RoboDK station: Tarea3Definitiva_IsabellaCeballos.rdk

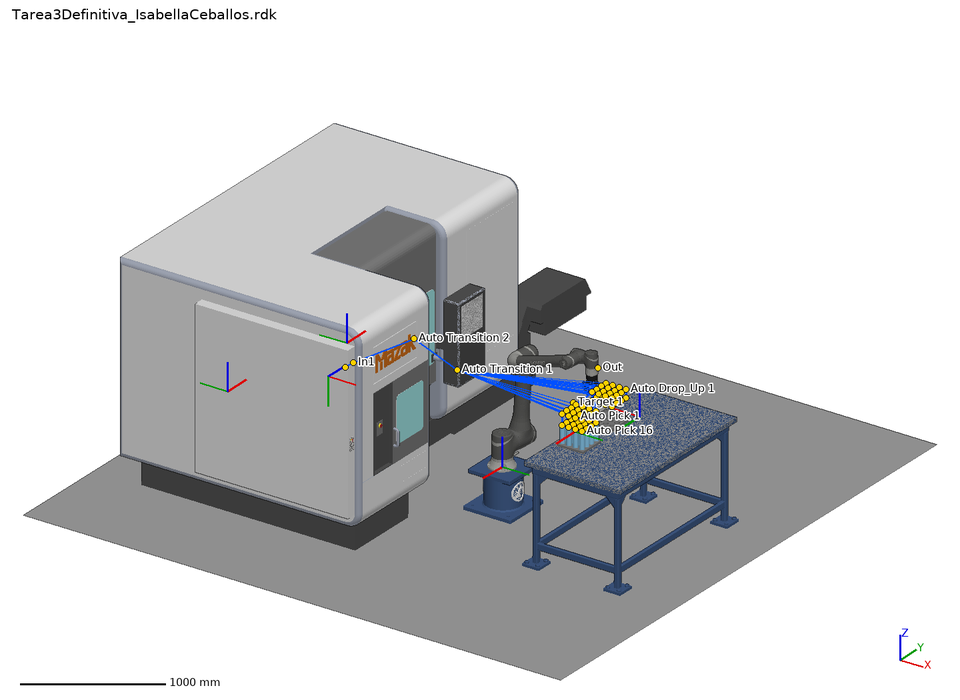
[picture v0: the station drawn from its stored meshes, robots at their saved joint values, targets as dots, program paths as lines]
Station Tarea3Definitiva_IsabellaCeballos (saved by RoboDK 5.5.1). Poses are relative to the parent item; angles as X-Y-Z fixed-axis rotations.
Station parameters (name, value as stored): TAGS, ['Machine Tending', 'CNC']
  - frame Omron TM12X Base at (300, 0, 70) mm, rotated rx 0 ry 0 rz -90 deg
    - robot Omron TM12X: 6 axes, payload 12 kg, reach 1300 mm, repeatability 0.1 mm, weight 33.3 kg
        modified DH rows (alpha deg, a mm, theta deg, d mm): 0, 0, 0, 165.2; 90, 0, 90, 0; 0, 636.1, 0, 0; 0, 557.9, -90, 156.3; -90, 0, 0, 106; 90, 0, 180, 113.15
        joint limits [-360, -360, -163, -360, -360, -360] to [360, 360, 163, 360, 360, 360]; home [0, 0, 90, -90, 90, 0]; saved at [263.092, -4.372, -66.936, -16.053, -91.349, 242.565]
      - tool g1, TCP at (0, 0, 130) mm, size 134.4 x 157.6 x 75 mm
      - tool RobotiQ 2F-85 Gripper (Open), TCP at (0, 0, 130) mm, size 147.4 x 146.8 x 75 mm
    - object Pedestal H12in (Type 1) at (0, 10, -300) mm, size 400 x 400 x 304.8 mm, geometry from Pedestal-H12in-Type-1.sld
  - frame Mazak Lathe Base at (-1000, 0, 650) mm, rotated rx 0 ry 0 rz 90 deg
    - robot Mazak Lathe: 1 axes
        modified DH rows (alpha deg, a mm, theta deg, d mm): 0, 0, 0, 0 linear
        base shift (0, 0, 0) mm, rotated rx 0 ry 90 rz 0 deg
        joint limits [0] to [700]; home [0]; saved at [0]
    - frame Lathe at (-368.68, -104.77, -79.13) mm, rotated rx -90 ry 0 rz -90 deg
  - frame Input at (1010, -140, 590) mm, rotated rx 0 ry 0 rz -90 deg
    - object Part Matrix at (0, 0, 0) mm, size 220 x 220 x 25 mm, geometry from Part Matrix.step
    - target Target 1 (Cartesian target) at (-26.53, -36.52, 202.61) mm, rotated rx -177.37 ry 1.91 rz -69.45 deg; joints [247.43, -1, -72.52, -13.29, -90.61, 226.91] of Omron TM12X
    - target Home (Cartesian target) at (28, 28, 225) mm, rotated rx -177.37 ry 1.91 rz -69.45 deg; joints [245.421, -8.702, -61.622, -16.467, -90.498, 224.904] of Omron TM12X
    - target Out (Cartesian target) at (-404.5, -94.61, 298.15) mm, rotated rx 179.32 ry 1.81 rz -82.53 deg; joints [279.536, -58.254, 58.657, -88.574, -89.388, -87.935] of Omron TM12X
    - target Auto Transition 1 (Cartesian target) at (259.07, -803.97, 350.52) mm, rotated rx -177.59 ry 1.72 rz -69.47 deg; joints [142.43, 16.067, -68.876, -37.376, -87.042, 121.929] of Omron TM12X
    - target Auto Transition 2 (Cartesian target) at (28.12, -1329.27, 350.52) mm, rotated rx -177.59 ry 1.72 rz -69.47 deg; joints [90.435, -6.151, -48.82, -37.474, -88.325, 69.903] of Omron TM12X
    - target Auto Up_Pick 1 (Cartesian target) at (28, 28, 225) mm, rotated rx -177.59 ry 1.72 rz -69.47 deg; joints [89.633, 54.83, -20.514, -126.784, -88.359, 69.101] of Omron TM12X
    - target Auto Pick 1 (Cartesian target) at (28, 28, 135) mm, rotated rx -177.59 ry 1.72 rz -69.47 deg; joints [89.633, 68.297, -42.42, -118.345, -88.359, 69.101] of Omron TM12X
    - target Auto Drop_Up 1 (Cartesian target) at (-374.01, 165.11, 220.31) mm, rotated rx -177.59 ry 1.72 rz -69.47 deg; joints [275.549, -61.889, 39.003, -64.828, -91.887, 255.015] of Omron TM12X
    - target Auto Drop 1 (Cartesian target) at (-374.01, 165.11, 156.87) mm, rotated rx -177.59 ry 1.72 rz -69.47 deg; joints [275.549, -69.478, 50.406, -68.642, -91.887, 255.015] of Omron TM12X
    - target Auto Up_Pick 2 (Cartesian target) at (28, 84, 225) mm, rotated rx -177.59 ry 1.72 rz -69.47 deg; joints [247.124, -65.005, 54.457, -76.543, -90.571, 226.613] of Omron TM12X
    - target Auto Pick 2 (Cartesian target) at (28, 84, 135) mm, rotated rx -177.59 ry 1.72 rz -69.47 deg; joints [89.659, 63.935, -29.058, -127.345, -88.358, 69.127] of Omron TM12X
    - target Auto Drop_Up 2 (Cartesian target) at (-374.01, 109.11, 220.31) mm, rotated rx -177.59 ry 1.72 rz -69.47 deg; joints [275.923, -64.235, 48.589, -72.079, -91.902, 255.389] of Omron TM12X
    - target Auto Drop 2 (Cartesian target) at (-374.01, 109.11, 156.87) mm, rotated rx -177.59 ry 1.72 rz -69.47 deg; joints [275.923, -71.126, 58.555, -75.154, -91.902, 255.389] of Omron TM12X
    - target Auto Up_Pick 3 (Cartesian target) at (28, 140, 225) mm, rotated rx -177.59 ry 1.72 rz -69.47 deg; joints [248.612, -20.473, -46.151, -20.483, -90.647, 228.099] of Omron TM12X
    - target Auto Pick 3 (Cartesian target) at (28, 140, 135) mm, rotated rx -177.59 ry 1.72 rz -69.47 deg; joints [248.612, -17.359, -60.205, -9.544, -90.647, 228.099] of Omron TM12X
    - target Auto Drop_Up 3 (Cartesian target) at (-374.01, 53.11, 220.31) mm, rotated rx -177.59 ry 1.72 rz -69.47 deg; joints [276.351, -13.266, -56.317, -18.157, -91.918, 255.817] of Omron TM12X
    - target Auto Drop 3 (Cartesian target) at (-374.01, 53.11, 156.87) mm, rotated rx -177.59 ry 1.72 rz -69.47 deg; joints [276.351, -11.379, -65.492, -10.869, -91.918, 255.817] of Omron TM12X
    - target Auto Up_Pick 4 (Cartesian target) at (28, 196, 225) mm, rotated rx -177.59 ry 1.72 rz -69.47 deg; joints [249.92, -27.448, -35.607, -24.068, -90.713, 229.405] of Omron TM12X
    - target Auto Pick 4 (Cartesian target) at (28, 196, 135) mm, rotated rx -177.59 ry 1.72 rz -69.47 deg; joints [249.92, -23.266, -51.89, -11.967, -90.713, 229.405] of Omron TM12X
    - target Auto Drop_Up 4 (Cartesian target) at (-374.01, -2.89, 220.31) mm, rotated rx -177.59 ry 1.72 rz -69.47 deg; joints [276.844, -7.931, -62.838, -16.988, -91.938, 256.31] of Omron TM12X
    - target Auto Drop 4 (Cartesian target) at (-374.01, -2.89, 156.87) mm, rotated rx -177.59 ry 1.72 rz -69.47 deg; joints [276.844, -6.251, -71.535, -9.971, -91.938, 256.31] of Omron TM12X
    - target Auto Up_Pick 5 (Cartesian target) at (84, 28, 225) mm, rotated rx -177.59 ry 1.72 rz -69.47 deg; joints [241.515, -10.232, -59.727, -17.09, -90.285, 221.011] of Omron TM12X
    - target Auto Pick 5 (Cartesian target) at (84, 28, 135) mm, rotated rx -177.59 ry 1.72 rz -69.47 deg; joints [241.515, -7.928, -72.043, -7.078, -90.285, 221.011] of Omron TM12X
    - target Auto Drop_Up 5 (Cartesian target) at (-318.01, 165.11, 220.31) mm, rotated rx -177.59 ry 1.72 rz -69.47 deg; joints [271.898, -23.816, -41.661, -22.121, -91.737, 251.365] of Omron TM12X
    - target Auto Drop 5 (Cartesian target) at (-318.01, 165.11, 156.87) mm, rotated rx -177.59 ry 1.72 rz -69.47 deg; joints [271.898, -21.097, -52.602, -13.899, -91.737, 251.365] of Omron TM12X
    - target Auto Up_Pick 6 (Cartesian target) at (84, 84, 225) mm, rotated rx -177.59 ry 1.72 rz -69.47 deg; joints [243.439, -15.802, -52.626, -18.633, -90.383, 222.933] of Omron TM12X
    - target Auto Pick 6 (Cartesian target) at (84, 84, 135) mm, rotated rx -177.59 ry 1.72 rz -69.47 deg; joints [243.439, -13.143, -65.721, -8.197, -90.383, 222.933] of Omron TM12X
    - target Auto Drop_Up 6 (Cartesian target) at (-318.01, 109.11, 220.31) mm, rotated rx -177.59 ry 1.72 rz -69.47 deg; joints [272.028, -17.436, -50.827, -19.34, -91.743, 251.496] of Omron TM12X
    - target Auto Drop 6 (Cartesian target) at (-318.01, 109.11, 156.87) mm, rotated rx -177.59 ry 1.72 rz -69.47 deg; joints [272.028, -15.303, -60.532, -11.766, -91.743, 251.496] of Omron TM12X
    - target Auto Up_Pick 7 (Cartesian target) at (84, 140, 225) mm, rotated rx -177.59 ry 1.72 rz -69.47 deg; joints [245.126, -21.925, -44.052, -21.096, -90.47, 224.618] of Omron TM12X
    - target Auto Pick 7 (Cartesian target) at (84, 140, 135) mm, rotated rx -177.59 ry 1.72 rz -69.47 deg; joints [245.126, -18.635, -58.475, -9.964, -90.47, 224.618] of Omron TM12X
    - target Auto Drop_Up 7 (Cartesian target) at (-318.01, 53.11, 220.31) mm, rotated rx -177.59 ry 1.72 rz -69.47 deg; joints [272.178, -11.695, -58.327, -17.585, -91.749, 251.645] of Omron TM12X
    - target Auto Drop 7 (Cartesian target) at (-318.01, 53.11, 156.87) mm, rotated rx -177.59 ry 1.72 rz -69.47 deg; joints [272.178, -9.884, -67.335, -10.387, -91.749, 251.645] of Omron TM12X
    - target Auto Up_Pick 8 (Cartesian target) at (84, 196, 225) mm, rotated rx -177.59 ry 1.72 rz -69.47 deg; joints [246.616, -29.108, -32.944, -25.035, -90.546, 226.106] of Omron TM12X
    - target Auto Pick 8 (Cartesian target) at (84, 196, 135) mm, rotated rx -177.59 ry 1.72 rz -69.47 deg; joints [246.616, -24.578, -49.957, -12.552, -90.546, 226.106] of Omron TM12X
    - target Auto Drop_Up 8 (Cartesian target) at (-318.01, -2.89, 220.31) mm, rotated rx -177.59 ry 1.72 rz -69.47 deg; joints [272.351, -6.333, -64.704, -16.575, -91.756, 251.819] of Omron TM12X
    - target Auto Drop 8 (Cartesian target) at (-318.01, -2.89, 156.87) mm, rotated rx -177.59 ry 1.72 rz -69.47 deg; joints [272.351, -4.699, -73.288, -9.625, -91.756, 251.819] of Omron TM12X
    - target Auto Up_Pick 9 (Cartesian target) at (140, 28, 225) mm, rotated rx -177.59 ry 1.72 rz -69.47 deg; joints [237.832, -12.037, -57.501, -17.499, -90.095, 217.333] of Omron TM12X
    - target Auto Pick 9 (Cartesian target) at (140, 28, 135) mm, rotated rx -177.59 ry 1.72 rz -69.47 deg; joints [237.832, -9.638, -70.034, -7.366, -90.095, 217.333] of Omron TM12X
    - target Auto Drop_Up 9 (Cartesian target) at (-262.01, 165.11, 220.31) mm, rotated rx -177.59 ry 1.72 rz -69.47 deg; joints [268.189, -22.573, -43.539, -21.379, -91.578, 247.658] of Omron TM12X
    - target Auto Drop 9 (Cartesian target) at (-262.01, 165.11, 156.87) mm, rotated rx -177.59 ry 1.72 rz -69.47 deg; joints [268.189, -19.996, -54.183, -13.312, -91.578, 247.658] of Omron TM12X
    - target Auto Up_Pick 10 (Cartesian target) at (140, 84, 225) mm, rotated rx -177.59 ry 1.72 rz -69.47 deg; joints [239.936, -17.62, -50.169, -19.254, -90.203, 219.434] of Omron TM12X
    - target Auto Pick 10 (Cartesian target) at (140, 84, 135) mm, rotated rx -177.59 ry 1.72 rz -69.47 deg; joints [239.936, -14.805, -63.596, -8.642, -90.203, 219.434] of Omron TM12X
    - target Auto Drop_Up 10 (Cartesian target) at (-262.01, 109.11, 220.31) mm, rotated rx -177.59 ry 1.72 rz -69.47 deg; joints [268.063, -16.266, -52.435, -18.786, -91.573, 247.532] of Omron TM12X
    - target Auto Drop 10 (Cartesian target) at (-262.01, 109.11, 156.87) mm, rotated rx -177.59 ry 1.72 rz -69.47 deg; joints [268.063, -14.216, -61.968, -11.304, -91.573, 247.532] of Omron TM12X
    - target Auto Up_Pick 11 (Cartesian target) at (140, 140, 225) mm, rotated rx -177.59 ry 1.72 rz -69.47 deg; joints [241.792, -23.852, -41.191, -22.008, -90.299, 221.288] of Omron TM12X
    - target Auto Pick 11 (Cartesian target) at (140, 140, 135) mm, rotated rx -177.59 ry 1.72 rz -69.47 deg; joints [241.792, -20.294, -56.173, -10.585, -90.299, 221.288] of Omron TM12X
    - target Auto Drop_Up 11 (Cartesian target) at (-262.01, 53.11, 220.31) mm, rotated rx -177.59 ry 1.72 rz -69.47 deg; joints [267.918, -10.535, -59.783, -17.165, -91.566, 247.387] of Omron TM12X
    - target Auto Drop 11 (Cartesian target) at (-262.01, 53.11, 156.87) mm, rotated rx -177.59 ry 1.72 rz -69.47 deg; joints [267.918, -8.774, -68.68, -10.029, -91.566, 247.387] of Omron TM12X
    - target Auto Up_Pick 12 (Cartesian target) at (140, 196, 225) mm, rotated rx -177.59 ry 1.72 rz -69.47 deg; joints [243.439, -31.4, -29.157, -26.504, -90.383, 222.933] of Omron TM12X
    - target Auto Pick 12 (Cartesian target) at (140, 196, 135) mm, rotated rx -177.59 ry 1.72 rz -69.47 deg; joints [243.439, -26.305, -47.355, -13.401, -90.383, 222.933] of Omron TM12X
    - target Auto Drop_Up 12 (Cartesian target) at (-262.01, -2.89, 220.31) mm, rotated rx -177.59 ry 1.72 rz -69.47 deg; joints [267.749, -5.144, -66.063, -16.272, -91.559, 247.219] of Omron TM12X
    - target Auto Drop 12 (Cartesian target) at (-262.01, -2.89, 156.87) mm, rotated rx -177.59 ry 1.72 rz -69.47 deg; joints [267.749, -3.538, -74.571, -9.369, -91.559, 247.219] of Omron TM12X
    - target Auto Up_Pick 13 (Cartesian target) at (196, 28, 225) mm, rotated rx -177.59 ry 1.72 rz -69.47 deg; joints [234.382, -14.253, -54.671, -18.113, -89.916, 213.888] of Omron TM12X
    - target Auto Pick 13 (Cartesian target) at (196, 28, 135) mm, rotated rx -177.59 ry 1.72 rz -69.47 deg; joints [234.382, -11.712, -67.515, -7.811, -89.916, 213.888] of Omron TM12X
    - target Auto Drop_Up 13 (Cartesian target) at (-206.01, 165.11, 220.31) mm, rotated rx -177.59 ry 1.72 rz -69.47 deg; joints [264.452, -21.782, -44.722, -20.889, -91.411, 243.923] of Omron TM12X
    - target Auto Drop 13 (Cartesian target) at (-206.01, 165.11, 156.87) mm, rotated rx -177.59 ry 1.72 rz -69.47 deg; joints [264.452, -19.29, -55.189, -12.914, -91.411, 243.923] of Omron TM12X
    - target Auto Up_Pick 14 (Cartesian target) at (196, 84, 225) mm, rotated rx -177.59 ry 1.72 rz -69.47 deg; joints [236.628, -19.883, -47.008, -20.145, -90.032, 216.131] of Omron TM12X
    - target Auto Pick 14 (Cartesian target) at (196, 84, 135) mm, rotated rx -177.59 ry 1.72 rz -69.47 deg; joints [236.628, -16.839, -60.917, -9.28, -90.032, 216.131] of Omron TM12X
    - target Auto Drop_Up 14 (Cartesian target) at (-206.01, 109.11, 220.31) mm, rotated rx -177.59 ry 1.72 rz -69.47 deg; joints [264.063, -15.515, -53.458, -18.41, -91.394, 243.534] of Omron TM12X
    - target Auto Drop 14 (Cartesian target) at (-206.01, 109.11, 156.87) mm, rotated rx -177.59 ry 1.72 rz -69.47 deg; joints [264.063, -13.514, -62.887, -10.982, -91.394, 243.534] of Omron TM12X
    - target Auto Up_Pick 15 (Cartesian target) at (196, 140, 225) mm, rotated rx -177.59 ry 1.72 rz -69.47 deg; joints [238.622, -26.311, -37.416, -23.312, -90.135, 218.122] of Omron TM12X
    - target Auto Pick 15 (Cartesian target) at (196, 140, 135) mm, rotated rx -177.59 ry 1.72 rz -69.47 deg; joints [238.622, -22.348, -53.243, -11.448, -90.135, 218.122] of Omron TM12X
    - target Auto Drop_Up 15 (Cartesian target) at (-206.01, 53.11, 220.31) mm, rotated rx -177.59 ry 1.72 rz -69.47 deg; joints [263.614, -9.785, -60.715, -16.873, -91.373, 243.087] of Omron TM12X
    - target Auto Drop 15 (Cartesian target) at (-206.01, 53.11, 156.87) mm, rotated rx -177.59 ry 1.72 rz -69.47 deg; joints [263.614, -8.054, -69.544, -9.775, -91.373, 243.087] of Omron TM12X
    - target Auto Up_Pick 16 (Cartesian target) at (196, 196, 225) mm, rotated rx -177.59 ry 1.72 rz -69.47 deg; joints [240.402, -34.545, -23.748, -28.751, -90.227, 219.899] of Omron TM12X
    - target Auto Pick 16 (Cartesian target) at (196, 196, 135) mm, rotated rx -177.59 ry 1.72 rz -69.47 deg; joints [240.402, -28.482, -43.987, -14.576, -90.227, 219.899] of Omron TM12X
    - target Auto Drop_Up 16 (Cartesian target) at (-206.01, -2.89, 220.31) mm, rotated rx -177.59 ry 1.72 rz -69.47 deg; joints [263.092, -4.372, -66.936, -16.053, -91.349, 242.565] of Omron TM12X
    - target Auto Drop 16 (Cartesian target) at (-206.01, -2.89, 156.87) mm, rotated rx -177.59 ry 1.72 rz -69.47 deg; joints [263.092, -2.783, -75.398, -9.18, -91.349, 242.565] of Omron TM12X
    - object Part 14 at (27.5, 137.5, -20) mm, size 40 x 40 x 150 mm, geometry from Part.step
    - object Part 13 at (27.5, 192.5, -20) mm, size 40 x 40 x 150 mm, geometry from Part.step
    - object Part 11 at (82.5, 82.5, -20) mm, size 40 x 40 x 150 mm, geometry from Part.step
    - object Part 10 at (82.5, 137.5, -20) mm, size 40 x 40 x 150 mm, geometry from Part.step
    - object Part 9 at (82.5, 192.5, -20) mm, size 40 x 40 x 150 mm, geometry from Part.step
    - object Part 8 at (137.5, 27.5, -20) mm, size 40 x 40 x 150 mm, geometry from Part.step
    - object Part 6 at (137.5, 137.5, -20) mm, size 40 x 40 x 150 mm, geometry from Part.step
    - object Part 1 at (192.5, 192.5, -20) mm, size 40 x 40 x 150 mm, geometry from Part.step
    - object Part 16 at (27.5, 27.5, -20) mm, size 40 x 40 x 150 mm, geometry from Part.step
    - object Part 12 at (82.5, 27.5, -20) mm, size 40 x 40 x 150 mm, geometry from Part.step
    - object Part 5 at (137.5, 192.5, -20) mm, size 40 x 40 x 150 mm, geometry from Part.step
    - object Part 7 at (137.5, 82.5, -20) mm, size 40 x 40 x 150 mm, geometry from Part.step
    - object Part 4 at (192.5, 27.5, -20) mm, rotated rx 0 ry 0 rz -180 deg, size 40 x 40 x 150 mm, geometry from Part.step
    - object Part 3 at (192.5, 82.5, -20) mm, rotated rx 0 ry 0 rz -180 deg, size 40 x 40 x 150 mm, geometry from Part.step
    - object Part 2 at (192.5, 137.5, -20) mm, rotated rx 0 ry 0 rz -180 deg, size 40 x 40 x 150 mm, geometry from Part.step
    - object Part 15 at (27.5, 82.5, -20) mm, size 40 x 40 x 150 mm, geometry from Part.step
  - frame Output at (1250, 290, 600) mm, rotated rx 0 ry 0 rz -180 deg
    - object Part Matrix at (47.8, 28.1, 0) mm, size 220 x 220 x 25 mm, geometry from Part Matrix.step
  - frame World at (-2000, 0, 0) mm, rotated rx 0 ry 0 rz 90 deg
    - object Floor at (250, -1940, -230) mm, size 4500 x 4500 x 0 mm, geometry from Floor (2).sld
    - object Table 1400x800x800mm at (-340, -3360, 570) mm, size 1420 x 820 x 800 mm, geometry from Table-1400x800x800mm.sld
    - target OpenDoor (Cartesian target) at (700, -1000, 650) mm; joints [700] of Mazak Lathe
    - target CloseDoor (Cartesian target) at (0, -1000, 650) mm; joints [0] of Mazak Lathe
    - target In1 (Cartesian target) at (-137.95, -1150.25, 595.88) mm, rotated rx -86.34 ry 2.11 rz 94.34 deg; joints [77.244, -89.992, 25.646, 51.981, -342.661, 170.292] of Omron TM12X
    - target In2 (Cartesian target) at (-206.56, -1130.76, 584.67) mm, rotated rx -87.8 ry 7.87 rz 92.76 deg; joints [-84.147, 66.082, 6.025, 75.079, -175.968, 40.623] of Omron TM12X
  - Python program Main_Program_Python (listed below)
  - program atach (1 instructions, listed below)
  - program detach (1 instructions, listed below)
  - program init (1 instructions, listed below)
  - program OpenDoor (2 instructions, listed below)
  - program CloseDoor (2 instructions, listed below)
  - program GoHome (3 instructions, listed below)
  - program Go_Out (3 instructions, listed below)
  - program Main_Program (496 instructions, listed below)
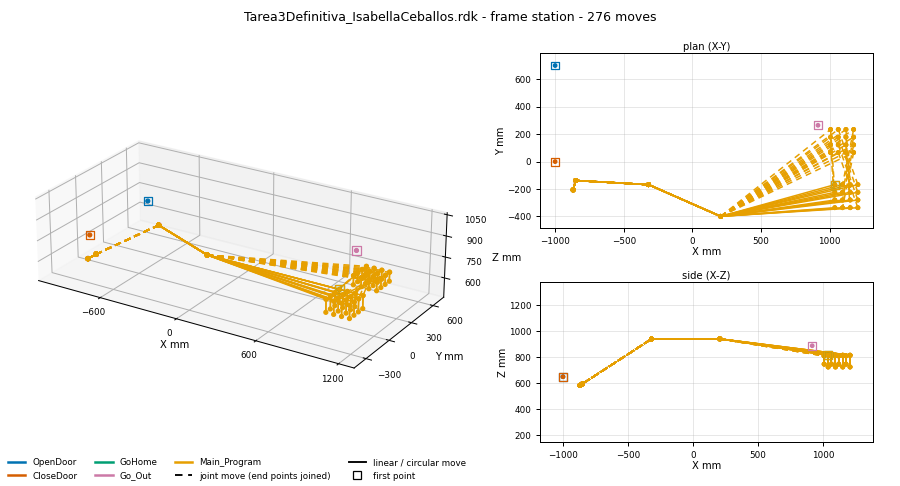
[picture p0: tool path of Tarea3Definitiva_IsabellaCeballos.rdk in frame station, 276 of 276 moves have a stored position in this frame; points joined in program order, loops and branches not executed]

--- Python program Main_Program_Python ---
from robolink import *    # Robot toolbox
import time as t

# Link to RoboDK
RDK = Robolink() # Interactuar con la interfaz del robot

# Mecanismos
robot = RDK.Item("Omron TM12X", ITEM_TYPE_ROBOT) #Robot
MAZAK = RDK.Item("Mazak Lathe") # Mazak
Tool_gripper = RDK.Item('g1',ITEM_TYPE_TOOL ) #Gripper

#Esto es para que no se repitan cosas en el código
list_names = RDK.ItemList(None, True)
for item_name in list_names:
    if item_name.startswith('Auto'):
        RDK.Item(item_name).Delete()
    if item_name.startswith('Main_'):
        RDK.Item(item_name).Delete()

#Código para generar puntos de botellas
def gridXY (m,n,d, e):

    """
     m= número de puntos en x
     n= número de puntos en y
     d= distancia entre cada punto en m

     En este ejercicio m = n, es cuadrado el soporte. 4x4
    """

    lista_puntos = []
    coeficientes = [1, 3, 5, 7 ]
    for i in range(m):
        for j in range(n):
            punto = [coeficientes[i]*d, coeficientes[j]*e, 225.000]
            lista_puntos.append(punto)


    return lista_puntos

m = 4
n = 4
d = 28
e = 28


puntos = gridXY(m,n,d,e)


# Código Principal

# Marcos de referencias
Input = RDK.Item("Input",ITEM_TYPE_FRAME) #frame
Output = RDK.Item("Output",ITEM_TYPE_FRAME)#frame2
Lathe = RDK.Item("Lathe",ITEM_TYPE_FRAME) #frame3
World = RDK.Item("World",ITEM_TYPE_FRAME) #frame4



robot.setPoseFrame(Input) #asociamos el robot a Input
pose_ref = robot.Pose()

Program = RDK.AddProgram('Main_Program')# Se genera programa


j = 0

#TARGETS DEL PROGRAMA

In1 = RDK.Item('In1',ITEM_TYPE_TARGET)
In2 = RDK.Item('In2',ITEM_TYPE_TARGET)
In3 = RDK.Item('In3',ITEM_TYPE_TARGET)


robot.setPoseFrame(Input)

    #TRANSITION 1
Trans1 = RDK.AddTarget('Auto Transition 1')#ti7
pose_t = pose_ref
pose_t.setPos([259.072, -803.965, 350.521] )
Trans1.setPose(pose_t)
Trans1.setAsCartesianTarget()
Trans1.setVisible(0)

    #TRANSITION 2
Trans2 = RDK.AddTarget('Auto Transition 2') #ti9
pose_t.setPos([28.119, -1329.271, 350.521] )
Trans2.setPose(pose_t)
Trans2.setAsCartesianTarget()
Trans2.setVisible(0)

# Funciones del programa

def Pick_up(P,Pick_Up,Pick):
    P.MoveJ(Pick_Up)
    t.sleep(0.5)
    P.MoveL(Pick)
    t.sleep(0.5)
    P.RunInstruction('atach',0)
    t.sleep(0.5)
    P.MoveL(Pick_Up)
    t.sleep(0.5)
    return

def Drop_out(P,Drop,Drop_Up):
    P.MoveJ(Drop_Up)
    t.sleep(0.5)
    P.MoveL(Drop)
    t.sleep(0.5)
    P.RunInstruction('detach',0)
    t.sleep(0.5)
    P.MoveL(Drop_Up)
    t.sleep(0.5)
    return

def Pick_Lathe_Transition(P,Trans1,Trans2):
    P.MoveL(Trans1)
    t.sleep(0.5)
    P.MoveJ(Trans2)
    t.sleep(0.5)
    return

def PickLathe(P,In1,In2,In3,Trans2):
    P.setFrame(World)
    P.MoveJ(In1)
    P.MoveL(In2)
    P.RunInstruction('detach',0)
    t.sleep(0.5)
    P.MoveL(In1)
    t.sleep(0.5)
    P.setFrame(Input)
    t.sleep(0.5)
    P.MoveJ(Trans2)
    t.sleep(5)
    return

def DropLathe(P,In1,In2,Trans2):
    P.setFrame(World)
    P.MoveJ(In1)
    P.MoveL(In2)
    P.RunInstruction('atach',0)
    t.sleep(0.5)
    P.MoveL(In1)
    t.sleep(0.5)
    P.setFrame(Input)
    t.sleep(0.5)
    P.MoveJ(Trans2)
    t.sleep(5)
    return


for i in puntos:

    #**GENARACIÓN DE TARGETS PICK BOTELLAS**
    #---------------------------------------
    robot.setPoseFrame(Input)
    Pick_Up = RDK.AddTarget('Auto Up_Pick %i' %(j+1))
    pose_i = pose_ref
    pose_i.setPos(i) #lista [x,y,z]
    Pick_Up.setPose(pose_i)
    Pick_Up.setAsCartesianTarget()
    Pick_Up.setVisible(0)
    #--------------------------------------
    Pick = RDK.AddTarget('Auto Pick %i' %(j+1))
    pose_j = pose_i
    pose_j.setPos([i[0],i[1], 135] )#[x,y,z]
    Pick.setPose(pose_j)
    Pick.setAsCartesianTarget()
    Pick.setVisible(0)



    #**GENERACIÓN DE TARGETS DROP BOTELLAS**
    #---------------------------------------
    Drop_Up = RDK.AddTarget('Auto Drop_Up %i' %(j+1))
    pose_p = pose_i
    pose_p.setPos([-402.010 + i[0], 193.114 - i[1], 220.306] )#[x,y,z]
    Drop_Up.setPose(pose_p)
    Drop_Up.setAsCartesianTarget()
    Drop_Up.setVisible(0)
   #---------------------------------------
    Drop = RDK.AddTarget('Auto Drop %i' %(j+1))
    pose_r = pose_i
    pose_r.setPos([-402.010 + i[0], 193.114 - i[1], 156.874] )#[x,y,z]
    Drop.setPose(pose_r)
    Drop.setAsCartesianTarget()
    Drop.setVisible(0)



    # SECUENCIA
    Program.setFrame(Input)
    Pick_up(Program,Pick_Up,Pick)
    Pick_Lathe_Transition(Program,Trans1,Trans2)
    Program.RunInstruction('OpenDoor',0)
    PickLathe(Program,In1,In2,In3,Trans2)
    Program.RunInstruction('CloseDoor',0)
    Program.RunInstruction('OpenDoor',0)
    DropLathe(Program,In1,In2,Trans2)
    Program.RunInstruction('CloseDoor',0)
    Program.MoveL(Trans1)
    Program.RunInstruction('Go_Out',0)
    Drop_out(Program,Drop,Drop_Up)


    j+=1

--- program atach (robot Omron TM12X) ---
  Adjuntar a g1

--- program detach (robot Omron TM12X) ---
  Separar de g1

--- program init (robot Omron TM12X) ---
  Reemplazar objetos

--- program OpenDoor (robot Mazak Lathe) ---
  Est. Ref.: World
  MoveJ (OpenDoor)

--- program CloseDoor (robot Mazak Lathe) ---
  Est. Ref.: World
  MoveJ (CloseDoor)

--- program GoHome (robot Omron TM12X) ---
  Est. Ref.: Input
  Est. herr: g1
  MoveJ (Home)

--- program Go_Out (robot Omron TM12X) ---
  Est. Ref.: Input
  Est. herr: g1
  MoveJ (Out)

--- program Main_Program (robot Omron TM12X) ---
  Est. Ref.: Input
  MoveJ (Auto Up_Pick 1)
  MoveL (Auto Pick 1)
  Llamar atach
  MoveL (Auto Up_Pick 1)
  MoveL (Auto Transition 1)
  MoveJ (Auto Transition 2)
  Llamar OpenDoor
  Est. Ref.: World
  MoveJ (In1)
  MoveL (In2)
  Llamar detach
  MoveL (In1)
  Est. Ref.: Input
  MoveJ (Auto Transition 2)
  Llamar CloseDoor
  Llamar OpenDoor
  Est. Ref.: World
  MoveJ (In1)
  MoveL (In2)
  Llamar atach
  MoveL (In1)
  Est. Ref.: Input
  MoveJ (Auto Transition 2)
  Llamar CloseDoor
  MoveL (Auto Transition 1)
  Llamar Go_Out
  MoveJ (Auto Drop_Up 1)
  MoveL (Auto Drop 1)
  Llamar detach
  MoveL (Auto Drop_Up 1)
  Est. Ref.: Input
  MoveJ (Auto Up_Pick 2)
  MoveL (Auto Pick 2)
  Llamar atach
  MoveL (Auto Up_Pick 2)
  MoveL (Auto Transition 1)
  MoveJ (Auto Transition 2)
  Llamar OpenDoor
  Est. Ref.: World
  MoveJ (In1)
  MoveL (In2)
  Llamar detach
  MoveL (In1)
  Est. Ref.: Input
  MoveJ (Auto Transition 2)
  Llamar CloseDoor
  Llamar OpenDoor
  Est. Ref.: World
  MoveJ (In1)
  MoveL (In2)
  Llamar atach
  MoveL (In1)
  Est. Ref.: Input
  MoveJ (Auto Transition 2)
  Llamar CloseDoor
  MoveL (Auto Transition 1)
  Llamar Go_Out
  MoveJ (Auto Drop_Up 2)
  MoveL (Auto Drop 2)
  Llamar detach
  MoveL (Auto Drop_Up 2)
  Est. Ref.: Input
  MoveJ (Auto Up_Pick 3)
  MoveL (Auto Pick 3)
  Llamar atach
  MoveL (Auto Up_Pick 3)
  MoveL (Auto Transition 1)
  MoveJ (Auto Transition 2)
  Llamar OpenDoor
  Est. Ref.: World
  MoveJ (In1)
  MoveL (In2)
  Llamar detach
  MoveL (In1)
  Est. Ref.: Input
  MoveJ (Auto Transition 2)
  Llamar CloseDoor
  Llamar OpenDoor
  Est. Ref.: World
  MoveJ (In1)
  MoveL (In2)
  Llamar atach
  MoveL (In1)
  Est. Ref.: Input
  MoveJ (Auto Transition 2)
  Llamar CloseDoor
  MoveL (Auto Transition 1)
  Llamar Go_Out
  MoveJ (Auto Drop_Up 3)
  MoveL (Auto Drop 3)
  Llamar detach
  MoveL (Auto Drop_Up 3)
  Est. Ref.: Input
  MoveJ (Auto Up_Pick 4)
  MoveL (Auto Pick 4)
  Llamar atach
  MoveL (Auto Up_Pick 4)
  MoveL (Auto Transition 1)
  MoveJ (Auto Transition 2)
  Llamar OpenDoor
  Est. Ref.: World
  MoveJ (In1)
  MoveL (In2)
  Llamar detach
  MoveL (In1)
  Est. Ref.: Input
  MoveJ (Auto Transition 2)
  Llamar CloseDoor
  Llamar OpenDoor
  Est. Ref.: World
  MoveJ (In1)
  MoveL (In2)
  Llamar atach
  MoveL (In1)
  Est. Ref.: Input
  MoveJ (Auto Transition 2)
  Llamar CloseDoor
  MoveL (Auto Transition 1)
  Llamar Go_Out
  MoveJ (Auto Drop_Up 4)
  MoveL (Auto Drop 4)
  Llamar detach
  MoveL (Auto Drop_Up 4)
  Est. Ref.: Input
  MoveJ (Auto Up_Pick 5)
  MoveL (Auto Pick 5)
  Llamar atach
  MoveL (Auto Up_Pick 5)
  MoveL (Auto Transition 1)
  MoveJ (Auto Transition 2)
  Llamar OpenDoor
  Est. Ref.: World
  MoveJ (In1)
  MoveL (In2)
  Llamar detach
  MoveL (In1)
  Est. Ref.: Input
  MoveJ (Auto Transition 2)
  Llamar CloseDoor
  Llamar OpenDoor
  Est. Ref.: World
  MoveJ (In1)
  MoveL (In2)
  Llamar atach
  MoveL (In1)
  Est. Ref.: Input
  MoveJ (Auto Transition 2)
  Llamar CloseDoor
  MoveL (Auto Transition 1)
  Llamar Go_Out
  MoveJ (Auto Drop_Up 5)
  MoveL (Auto Drop 5)
  Llamar detach
  MoveL (Auto Drop_Up 5)
  Est. Ref.: Input
  MoveJ (Auto Up_Pick 6)
  MoveL (Auto Pick 6)
  Llamar atach
  MoveL (Auto Up_Pick 6)
  MoveL (Auto Transition 1)
  MoveJ (Auto Transition 2)
  Llamar OpenDoor
  Est. Ref.: World
  MoveJ (In1)
  MoveL (In2)
  Llamar detach
  MoveL (In1)
  Est. Ref.: Input
  MoveJ (Auto Transition 2)
  Llamar CloseDoor
  Llamar OpenDoor
  Est. Ref.: World
  MoveJ (In1)
  MoveL (In2)
  Llamar atach
  MoveL (In1)
  Est. Ref.: Input
  MoveJ (Auto Transition 2)
  Llamar CloseDoor
  MoveL (Auto Transition 1)
  Llamar Go_Out
  MoveJ (Auto Drop_Up 6)
  MoveL (Auto Drop 6)
  Llamar detach
  MoveL (Auto Drop_Up 6)
  Est. Ref.: Input
  MoveJ (Auto Up_Pick 7)
  MoveL (Auto Pick 7)
  Llamar atach
  MoveL (Auto Up_Pick 7)
  MoveL (Auto Transition 1)
  MoveJ (Auto Transition 2)
  Llamar OpenDoor
  Est. Ref.: World
  MoveJ (In1)
  MoveL (In2)
  Llamar detach
  MoveL (In1)
  Est. Ref.: Input
  MoveJ (Auto Transition 2)
  Llamar CloseDoor
  Llamar OpenDoor
  Est. Ref.: World
  MoveJ (In1)
  MoveL (In2)
  Llamar atach
  MoveL (In1)
  Est. Ref.: Input
  MoveJ (Auto Transition 2)
  Llamar CloseDoor
  MoveL (Auto Transition 1)
  Llamar Go_Out
  MoveJ (Auto Drop_Up 7)
  MoveL (Auto Drop 7)
  Llamar detach
  MoveL (Auto Drop_Up 7)
  Est. Ref.: Input
  MoveJ (Auto Up_Pick 8)
  MoveL (Auto Pick 8)
  Llamar atach
  MoveL (Auto Up_Pick 8)
  MoveL (Auto Transition 1)
  MoveJ (Auto Transition 2)
  Llamar OpenDoor
  Est. Ref.: World
  MoveJ (In1)
  MoveL (In2)
  Llamar detach
  MoveL (In1)
  Est. Ref.: Input
  MoveJ (Auto Transition 2)
  Llamar CloseDoor
  Llamar OpenDoor
  Est. Ref.: World
  MoveJ (In1)
  MoveL (In2)
  Llamar atach
  MoveL (In1)
  Est. Ref.: Input
  MoveJ (Auto Transition 2)
  Llamar CloseDoor
  MoveL (Auto Transition 1)
  Llamar Go_Out
  MoveJ (Auto Drop_Up 8)
  MoveL (Auto Drop 8)
  Llamar detach
  MoveL (Auto Drop_Up 8)
  Est. Ref.: Input
  MoveJ (Auto Up_Pick 9)
  MoveL (Auto Pick 9)
  Llamar atach
  MoveL (Auto Up_Pick 9)
  MoveL (Auto Transition 1)
  MoveJ (Auto Transition 2)
  Llamar OpenDoor
  Est. Ref.: World
  MoveJ (In1)
  MoveL (In2)
  Llamar detach
  MoveL (In1)
  Est. Ref.: Input
  MoveJ (Auto Transition 2)
  Llamar CloseDoor
  Llamar OpenDoor
  Est. Ref.: World
  MoveJ (In1)
  MoveL (In2)
  Llamar atach
  MoveL (In1)
  Est. Ref.: Input
  MoveJ (Auto Transition 2)
  Llamar CloseDoor
  MoveL (Auto Transition 1)
  Llamar Go_Out
  MoveJ (Auto Drop_Up 9)
  MoveL (Auto Drop 9)
  Llamar detach
  MoveL (Auto Drop_Up 9)
  Est. Ref.: Input
  MoveJ (Auto Up_Pick 10)
  MoveL (Auto Pick 10)
  Llamar atach
  MoveL (Auto Up_Pick 10)
  MoveL (Auto Transition 1)
  MoveJ (Auto Transition 2)
  Llamar OpenDoor
  Est. Ref.: World
  MoveJ (In1)
  MoveL (In2)
  Llamar detach
  MoveL (In1)
  Est. Ref.: Input
  MoveJ (Auto Transition 2)
  Llamar CloseDoor
  Llamar OpenDoor
  Est. Ref.: World
  MoveJ (In1)
  MoveL (In2)
  Llamar atach
  MoveL (In1)
  Est. Ref.: Input
  MoveJ (Auto Transition 2)
  Llamar CloseDoor
  MoveL (Auto Transition 1)
  Llamar Go_Out
  MoveJ (Auto Drop_Up 10)
  MoveL (Auto Drop 10)
  Llamar detach
  MoveL (Auto Drop_Up 10)
  Est. Ref.: Input
  MoveJ (Auto Up_Pick 11)
  MoveL (Auto Pick 11)
  Llamar atach
  MoveL (Auto Up_Pick 11)
  MoveL (Auto Transition 1)
  MoveJ (Auto Transition 2)
  Llamar OpenDoor
  Est. Ref.: World
  MoveJ (In1)
  MoveL (In2)
  Llamar detach
  MoveL (In1)
  Est. Ref.: Input
  MoveJ (Auto Transition 2)
  Llamar CloseDoor
  Llamar OpenDoor
  Est. Ref.: World
  MoveJ (In1)
  MoveL (In2)
  Llamar atach
  MoveL (In1)
  Est. Ref.: Input
  MoveJ (Auto Transition 2)
  Llamar CloseDoor
  MoveL (Auto Transition 1)
  Llamar Go_Out
  MoveJ (Auto Drop_Up 11)
  MoveL (Auto Drop 11)
  Llamar detach
  MoveL (Auto Drop_Up 11)
  Est. Ref.: Input
  MoveJ (Auto Up_Pick 12)
  MoveL (Auto Pick 12)
  Llamar atach
  MoveL (Auto Up_Pick 12)
  MoveL (Auto Transition 1)
  MoveJ (Auto Transition 2)
  Llamar OpenDoor
  Est. Ref.: World
  MoveJ (In1)
  MoveL (In2)
  Llamar detach
  MoveL (In1)
  Est. Ref.: Input
  MoveJ (Auto Transition 2)
  Llamar CloseDoor
  Llamar OpenDoor
  Est. Ref.: World
  MoveJ (In1)
  MoveL (In2)
  Llamar atach
  MoveL (In1)
  Est. Ref.: Input
  MoveJ (Auto Transition 2)
  Llamar CloseDoor
  MoveL (Auto Transition 1)
  Llamar Go_Out
  MoveJ (Auto Drop_Up 12)
  MoveL (Auto Drop 12)
  Llamar detach
  MoveL (Auto Drop_Up 12)
  Est. Ref.: Input
  MoveJ (Auto Up_Pick 13)
  MoveL (Auto Pick 13)
  Llamar atach
  MoveL (Auto Up_Pick 13)
  MoveL (Auto Transition 1)
  MoveJ (Auto Transition 2)
  Llamar OpenDoor
  Est. Ref.: World
  MoveJ (In1)
  MoveL (In2)
  Llamar detach
  MoveL (In1)
  Est. Ref.: Input
  MoveJ (Auto Transition 2)
  Llamar CloseDoor
  Llamar OpenDoor
  Est. Ref.: World
  MoveJ (In1)
  MoveL (In2)
  Llamar atach
  MoveL (In1)
  Est. Ref.: Input
  MoveJ (Auto Transition 2)
  Llamar CloseDoor
  MoveL (Auto Transition 1)
  Llamar Go_Out
  MoveJ (Auto Drop_Up 13)
  MoveL (Auto Drop 13)
  Llamar detach
  MoveL (Auto Drop_Up 13)
  Est. Ref.: Input
  MoveJ (Auto Up_Pick 14)
  MoveL (Auto Pick 14)
  Llamar atach
  MoveL (Auto Up_Pick 14)
  MoveL (Auto Transition 1)
  MoveJ (Auto Transition 2)
  Llamar OpenDoor
  Est. Ref.: World
  MoveJ (In1)
  MoveL (In2)
  Llamar detach
  MoveL (In1)
  Est. Ref.: Input
  MoveJ (Auto Transition 2)
  Llamar CloseDoor
  Llamar OpenDoor
  Est. Ref.: World
  MoveJ (In1)
  MoveL (In2)
  Llamar atach
  MoveL (In1)
  Est. Ref.: Input
  MoveJ (Auto Transition 2)
  Llamar CloseDoor
  MoveL (Auto Transition 1)
  Llamar Go_Out
  MoveJ (Auto Drop_Up 14)
  MoveL (Auto Drop 14)
  Llamar detach
  MoveL (Auto Drop_Up 14)
  Est. Ref.: Input
  MoveJ (Auto Up_Pick 15)
  MoveL (Auto Pick 15)
  Llamar atach
  MoveL (Auto Up_Pick 15)
  MoveL (Auto Transition 1)
  MoveJ (Auto Transition 2)
  Llamar OpenDoor
  Est. Ref.: World
  MoveJ (In1)
  MoveL (In2)
  Llamar detach
  MoveL (In1)
  Est. Ref.: Input
  MoveJ (Auto Transition 2)
  Llamar CloseDoor
  Llamar OpenDoor
  Est. Ref.: World
  MoveJ (In1)
  MoveL (In2)
  Llamar atach
  MoveL (In1)
  Est. Ref.: Input
  MoveJ (Auto Transition 2)
  Llamar CloseDoor
  MoveL (Auto Transition 1)
  Llamar Go_Out
  MoveJ (Auto Drop_Up 15)
  MoveL (Auto Drop 15)
  Llamar detach
  MoveL (Auto Drop_Up 15)
  Est. Ref.: Input
  MoveJ (Auto Up_Pick 16)
  MoveL (Auto Pick 16)
  Llamar atach
  MoveL (Auto Up_Pick 16)
  MoveL (Auto Transition 1)
  MoveJ (Auto Transition 2)
  Llamar OpenDoor
  Est. Ref.: World
  MoveJ (In1)
  MoveL (In2)
  Llamar detach
  MoveL (In1)
  Est. Ref.: Input
  MoveJ (Auto Transition 2)
  Llamar CloseDoor
  Llamar OpenDoor
  Est. Ref.: World
  MoveJ (In1)
  MoveL (In2)
  Llamar atach
  MoveL (In1)
  Est. Ref.: Input
  MoveJ (Auto Transition 2)
  Llamar CloseDoor
  MoveL (Auto Transition 1)
  Llamar Go_Out
  MoveJ (Auto Drop_Up 16)
  MoveL (Auto Drop 16)
  Llamar detach
  MoveL (Auto Drop_Up 16)
